// TIA Portal V21 export
FUNCTION "GestLampallarmeRGY" : Void   // FC28, LAD
{ S7_Optimized_Access := 'TRUE' }
// stored: SetENOAutomatically false
   VAR_INPUT
      K_Zona : Int;
   END_VAR
   VAR_OUTPUT
      R : Bool;   // Uscita colore Red
      G : Bool;   // Uscita colore Green
      Y : Bool;   // Uscita colore Yellow
   END_VAR
   VAR_TEMP
      LampeggioVerde : Bool;
      VerdeFisso : Bool;
      LampeggioRosso : Bool;
      GialloLampeggiante : Bool;
      GialloFisso : Bool;
      UtenzeInMan : Bool;
      CounterUtenze : Int;
   END_VAR
BEGIN

REGION Network 1 (SCL)
   #UtenzeInMan := False;
   FOR #CounterUtenze := 0 TO "K_NumValvola" DO
       IF "Valvola".V[#CounterUtenze].Rif_Inc.K_Zona = #K_Zona THEN
           IF NOT ("Valvola".V[#CounterUtenze].Out.Stato = 0 OR "Valvola".V[#CounterUtenze].Out.Stato = 2) THEN
               #UtenzeInMan := True;
           END_IF;
       END_IF;
   END_FOR;
   FOR #CounterUtenze := 0 TO "K_NumMotore" DO
       IF "Motore".M[#CounterUtenze].Rif_Inc.K_Zona = #K_Zona THEN
           IF NOT ("Motore".M[#CounterUtenze].HMI.Stato = 0 OR "Valvola".V[#CounterUtenze].Out.Stato = 1) THEN
               #UtenzeInMan := True;
           END_IF;
       END_IF;
   END_FOR;

   #LampeggioRosso := "Zona".Z[#K_Zona].Out.CumulativoAllarmi;
   #VerdeFisso := "Zona".Z[#K_Zona].Out.Auto;
   #LampeggioVerde := ("Zona".Z[#K_Zona].Out.Man OR #UtenzeInMan) OR (#VerdeFisso AND #LampeggioRosso);
   #GialloFisso := "Zona".Z[#K_Zona].Out.Attesa;
   #GialloLampeggiante := #GialloFisso AND #LampeggioRosso;
END_REGION

REGION Network 2: Uscita colore Red
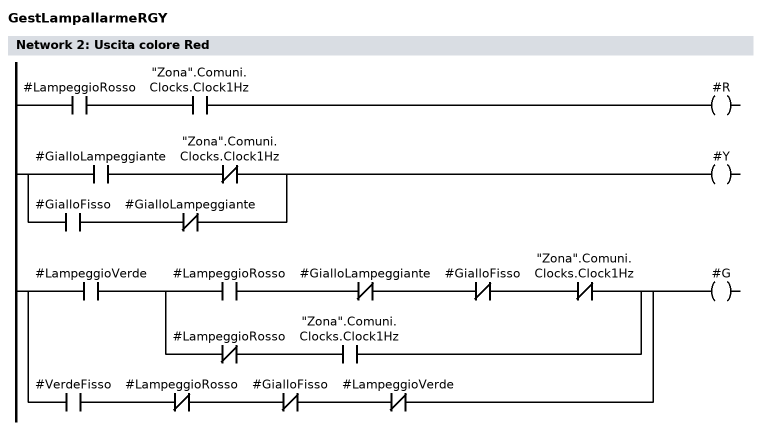
   RUNG wire#powerrail
      Contact( #LampeggioRosso )
      Contact( "Zona".Comuni.Clocks.Clock1Hz )
      Coil( #R )
   END_RUNG
   RUNG wire#powerrail
      Contact( #GialloLampeggiante )
      I_Contact( "Zona".Comuni.Clocks.Clock1Hz )
      wire#w1
      Coil( #Y )
   END_RUNG
   RUNG wire#powerrail
      Contact( #GialloFisso )
      I_Contact( #GialloLampeggiante )
   END_RUNG wire#w1
   RUNG wire#powerrail
      Contact( #LampeggioVerde )
      wire#w2
      Contact( #LampeggioRosso )
      I_Contact( #GialloLampeggiante )
      I_Contact( #GialloFisso )
      I_Contact( "Zona".Comuni.Clocks.Clock1Hz )
      wire#w3
      Coil( #G )
   END_RUNG
   RUNG wire#w2
      I_Contact( #LampeggioRosso )
      Contact( "Zona".Comuni.Clocks.Clock1Hz )
   END_RUNG wire#w3
   RUNG wire#powerrail
      Contact( #VerdeFisso )
      I_Contact( #LampeggioRosso )
      I_Contact( #GialloFisso )
      I_Contact( #LampeggioVerde )
   END_RUNG wire#w3
   // the same network as SCL:
   #R := #LampeggioRosso AND "Zona".Comuni.Clocks.Clock1Hz;
   #Y := (#GialloLampeggiante AND NOT "Zona".Comuni.Clocks.Clock1Hz) OR (#GialloFisso AND NOT #GialloLampeggiante);
   #G := (#LampeggioVerde AND ((#LampeggioRosso AND NOT #GialloLampeggiante AND NOT #GialloFisso AND NOT "Zona".Comuni.Clocks.Clock1Hz) OR (NOT #LampeggioRosso AND "Zona".Comuni.Clocks.Clock1Hz))) OR (#VerdeFisso AND NOT #LampeggioRosso AND NOT #GialloFisso AND NOT #LampeggioVerde);
END_REGION
END_FUNCTION
